// TIA Portal project "SCL CALCULADORA" (V11)

(* hardware
DEVICE "S7300/ET200 station_1"  SIMATIC 300-Station
   slot 0: "Perfil soporte_0"  Rail  6ES7 390-1***0-0AA0
   slot 2: "PLC_1"  CPU 313C-2 DP  6ES7 313-6CF03-0AB0  V2.6
      slot 0: "Interfaz MPI_1"  MPI
      slot 1: "Interfaz DP_1"  DP
      slot 2: "DI16/DO16_1"  DI16/DO16
      slot 4: "Contaje_1"  Counter
*)

// ===== PLC "PLC_1"  CPU 313C-2 DP =====

VAR_GLOBAL   // PLC tag table "Tabla de variables estándar"
   "Tag_1" AT %MD0 : Real;
   "Tag_2" AT %E0.0 : Bool;
   "Tag_3" AT %E0.1 : Bool;
   "Tag_4" AT %E0.2 : Bool;
   "Tag_5" AT %E0.3 : Bool;
   "Tag_6" AT %E0.4 : Bool;
   "Tag_7" AT %E0.5 : Bool;
   "Tag_8" AT %E0.6 : Bool;
   "Tag_9" AT %E1.0 : Bool;
   "Tag_10" AT %E1.1 : Bool;
   "Tag_11" AT %E1.2 : Bool;
   "Tag_12" AT %E1.3 : Bool;
   "Tag_13" AT %E1.4 : Bool;
   "Tag_14" AT %E1.5 : Bool;
   "Tag_15" AT %E1.6 : Bool;
   "Tag_16" AT %E1.7 : Bool;
   "Tag_17" AT %E2.0 : Bool;
   "Tag_18" AT %E2.1 : Bool;
   "Tag_19" AT %E0.7 : Bool;
   "Tag_20" AT %M0.0 : Bool;
   "Tag_21" AT %E2.2 : Bool;
   "Tag_22" AT %E2.3 : Bool;
   "Tag_23" AT %E2.4 : Bool;
   "Tag_24" AT %MD4 : Real;
   "Tag_25" AT %A0.0 : Bool;
   "Tag_26" AT %E2.7 : Bool;
   "Tag_27" AT %MD8 : Real;
   "Tag_28" AT %MD12 : Real;
   "Tag_29" AT %MD16 : Real;
   "Tag_30" AT %MD20 : Real;
   "Tag_31" AT %MD24 : Real;
   "Tag_32" AT %MD28 : Real;
   "Tag_33" AT %MD32 : Real;
   "Tag_34" AT %MD36 : Real;
   "Tag_35" AT %MD40 : Real;
   "Tag_36" AT %MD44 : Real;
   "Tag_37" AT %MD48 : Real;
   "Tag_38" AT %MD52 : Real;
   "Tag_39" AT %MD56 : Real;
   "Tag_40" AT %MD60 : Real;
   "Tag_41" AT %MD64 : Real;
   "Tag_42" AT %E2.5 : Bool;
END_VAR

DATA_BLOCK "CALCULADORA_DB"   // DB1
{ S7_Optimized_Access := 'FALSE' }
VERSION : 0.1
// stored: InstanceOfName CALCULADORA
"CALCULADORA"
BEGIN
END_DATA_BLOCK

FUNCTION_BLOCK "CALCULADORA"   // FB1, SCL
{ S7_Optimized_Access := 'FALSE' }
VERSION : 0.1
   VAR_INPUT
      "N º 1" : Bool;
      "N º 2" : Bool;
      "N º 3" : Bool;
      "N º 4" : Bool;
      "N º 5" : Bool;
      "N º 6" : Bool;
      "N º 7" : Bool;
      "N º 8" : Bool;
      "N º 9" : Bool;
      "N º 0" : Bool;
      "TECLA +" : Bool;
      "TECLA -" : Bool;
      "TECLA *" : Bool;
      "TECLA /" : Bool;
      CE : Bool;
      C : Bool;
      "TECLA =" : Bool;
      "TECLA +/-" : Bool;
      COMA : Bool;
      Min : Bool;
      MR : Bool;
      "RAIZ CUADRADA" : Bool;
   END_VAR
   VAR_OUTPUT
      RESULTADO : Real;
   END_VAR
   VAR
      CONTAJE : Int;
      "A" : Int;
      "CONTAJE +/-" : Int;
      "A +/-" : Int;
      M0 : Bool;
      M1 : Bool;
      M2 : Bool;
      M3 : Bool;
      M4 : Bool;
      M5 : Bool;
      M6 : Bool;
      M7 : Bool;
      M8 : Bool;
      M9 : Bool;
      M10 : Bool;
      M11 : Bool;
      M12 : Bool;
      M13 : Bool;
      M14 : Bool;
      M15 : Bool;
      M16 : Bool;
      M17 : Bool;
      M18 : Bool;
      M19 : Bool;
      T0 : Bool;
      "Nº 10" : Real := 10.0;
      Nº100 : Real := 100.0;
      Nº1000 : Real := 1000.0;
      Nº10000 : Real := 10000.0;
      Nº100000 : Real := 100000.0;
      Nº1000000 : Real := 1000000.0;
      "ORDEN A" : Real;
      "ORDEN B" : Real;
      "ORDEN X/10" : Real;
      "ORDEN X/100" : Real;
      "ORDEN X/1000" : Real;
      "ORDEN X/10000" : Real;
      "ORDEN X/100000" : Real;
      "ORDEN X/1000000" : Real;
      "OPERANDO 1" : Real;
      ACUMULATIVO : Real;
      "X 1" : Real;
      "X 10" : Real;
      "X 100" : Real;
      "X 1000" : Real;
      "X 10000" : Real;
      "X 100000" : Real;
      "X/10" : Real := 10.0;
      "X/100" : Real := 100.0;
      "X/1000" : Real := 1000.0;
      "X/10000" : Real := 10000.0;
      "X/100000" : Real := 100000.0;
      "X/1000000" : Real := 1000000.0;
      MEMORIA : Real;
      VISUALIZAR : Time;
   END_VAR
BEGIN
END_FUNCTION_BLOCK

ORGANIZATION_BLOCK "Main"   // OB1, LAD
TITLE = "Main Program Sweep (Cycle)"
{ S7_Optimized_Access := 'FALSE' }
VERSION : 0.1
   VAR_TEMP
      OB1_EV_CLASS : Byte;   // Bits 0-3 = 1 (Coming event), Bits 4-7 = 1 (Event class 1)
      OB1_SCAN_1 : Byte;   // 1 (Cold restart scan 1 of OB 1), 3 (Scan 2-n of OB 1)
      OB1_PRIORITY : Byte;   // Priority of OB Execution
      OB1_OB_NUMBR : Byte;   // 1 (Organization block 1, OB1)
      OB1_RESERVED_1 : Byte;   // Reserved for system
      OB1_RESERVED_2 : Byte;   // Reserved for system
      OB1_PREV_CYCLE : Int;   // Cycle time of previous OB1 scan (milliseconds)
      OB1_MIN_CYCLE : Int;   // Minimum cycle time of OB1 (milliseconds)
      OB1_MAX_CYCLE : Int;   // Maximum cycle time of OB1 (milliseconds)
      OB1_DATE_TIME : Date_And_Time;   // Date and time OB1 started
   END_VAR
BEGIN

REGION Network 1
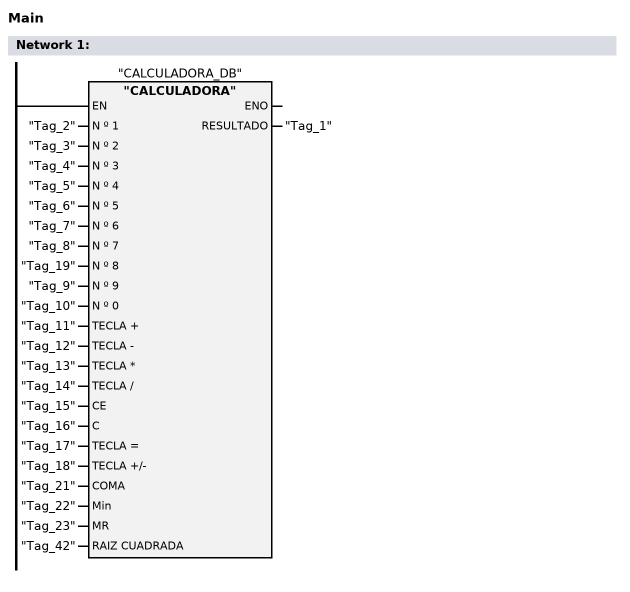
   RUNG wire#powerrail
      "CALCULADORA_DB"("N º 1" := "Tag_2", "N º 2" := "Tag_3", "N º 3" := "Tag_4", "N º 4" := "Tag_5", "N º 5" := "Tag_6", "N º 6" := "Tag_7", "N º 7" := "Tag_8", "N º 8" := "Tag_19", "N º 9" := "Tag_9", "N º 0" := "Tag_10", "TECLA +" := "Tag_11", "TECLA -" := "Tag_12", "TECLA *" := "Tag_13", "TECLA /" := "Tag_14", CE := "Tag_15", C := "Tag_16", "TECLA =" := "Tag_17", "TECLA +/-" := "Tag_18", COMA := "Tag_21", Min := "Tag_22", MR := "Tag_23", "RAIZ CUADRADA" := "Tag_42", RESULTADO => "Tag_1")
   END_RUNG
   // the same network as SCL:
   "CALCULADORA_DB"("N º 1" := "Tag_2",   // "CALCULADORA"
                    "N º 2" := "Tag_3",
                    "N º 3" := "Tag_4",
                    "N º 4" := "Tag_5",
                    "N º 5" := "Tag_6",
                    "N º 6" := "Tag_7",
                    "N º 7" := "Tag_8",
                    "N º 8" := "Tag_19",
                    "N º 9" := "Tag_9",
                    "N º 0" := "Tag_10",
                    "TECLA +" := "Tag_11",
                    "TECLA -" := "Tag_12",
                    "TECLA *" := "Tag_13",
                    "TECLA /" := "Tag_14",
                    CE := "Tag_15",
                    C := "Tag_16",
                    "TECLA =" := "Tag_17",
                    "TECLA +/-" := "Tag_18",
                    COMA := "Tag_21",
                    Min := "Tag_22",
                    MR := "Tag_23",
                    "RAIZ CUADRADA" := "Tag_42",
                    RESULTADO => "Tag_1");
END_REGION
END_ORGANIZATION_BLOCK